Omron CX-Programmer project NewProject (CX-Programmer 9.51)

# PLC NewPLC1: CP1L L

## Program NewProgram1 (cyclic task 0)
Local symbols
przycisk_start 0.05 BOOL  ; Start grzałki

### Section Section1

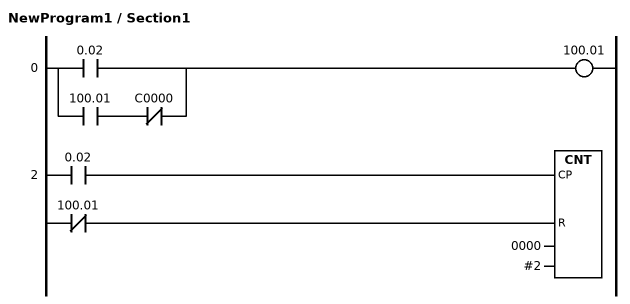
; rung 0
LD 0.02
LD 100.01
ANDNOT C0000
ORLD
OUT 100.01
; rung 2
LD 0.02
LDNOT 100.01
CNT 0000 #2

### Section END
; rung 0
END(001)